FUNCTION_BLOCK F_SHR (* bitwise shift right function *)
  PACKAGE iec61131::bitwiseOperators;
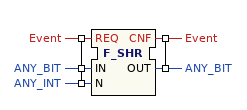
  EVENT_INPUT
    REQ WITH IN, N; (* Service Request *)
  END_EVENT
  EVENT_OUTPUT
    CNF WITH OUT; (* Confirmation of Requested Service *)
  END_EVENT
  VAR_INPUT
    IN : ANY_BIT; (* right-shifted *)
    N : ANY_INT; (* right-shifted by N bits *)
  END_VAR
  VAR_OUTPUT
    OUT : ANY_BIT; (* right-shifted by N zero-filled on left *)
  END_VAR
END_FUNCTION_BLOCK
